FUNCTION_BLOCK FB_CO_ABERRATION
VAR_INPUT
	jd			: LREAL;		// Julian Date
	ra			: LREAL;		// RA in degrees
	dec			: LREAL; 		// Dec in degrees
	eps 		: LREAL := 0.0;
END_VAR
VAR_OUTPUT
	d_ra		: LREAL;
	d_dec		: LREAL;
END_VAR
VAR
	sunpos		: FB_SUNPOS;
	nutate		: FB_IAU2000B;
	sunra		: LREAL;
	sundec		: LREAL;
	sunlon		: LREAL;
	d_psi		: LREAL;
	d_epsilon	: LREAL; 
	eps_loc		: LREAL;		// obliquity in radians, eps or calculated if eps = 0
	t, e, peri, cd, sd, ce, te, cp, sp, cs, ss, ca, sa, term1, term2, term3, term4: LREAL;
END_VAR
VAR CONSTANT
	d2r 		: LREAL := PI/180.0;
	k			: LREAL := 20.49552; 	//constant of aberration, in arcseconds
	
END_VAR

(* https://github.com/wlandsman/IDLAstro/blob/master/pro/co_aberration.pro
;+
;  NAME:
;     CO_ABERRATION
; PURPOSE:
;     Calculate changes to Ra and Dec due to the effect of annual aberration 
; EXPLANATION:
;      as described in Meeus, Chap 23.
; CALLING SEQUENCE:
;      co_aberration, jd, ra, dec, d_ra, d_dec, [EPS = ]
; INPUTS
;       jd      : Julian Date [scalar or vector]
;       ra, dec : ra  and dec's in degrees
;
; OUTPUTS
;       d_ra, d_dec: the corrections to ra and dec due to aberration in 
;                    degrees.  (These values can be added to the true RA 
;                    and dec to get the apparent position).   Note that d_ra
;                     is *not* multiplied by cos(dec), so that 
;                     apparent_ra = ra + d_ra. 
; OPTIONAL INPUT KEYWORD:
;       eps : set this to the true obliquity of the ecliptic (in radians), or
;         it will be set for you if you don't know it (in that case, set it to
;                 an empty variable).
; NOTES:
;  These formula are from Meeus, Chapters 23.  Accuracy is much better than 1 
;   arcsecond.
;
;   The maximum deviation due to annual aberration is 20.49" and occurs when the
;   Earth velocity is perpendicular to the direction of the star.
;
; REVISION HISTORY:
;   Written, June 2002,      Chris O'Dell, U. of Wisconsin
;   Fix error with vector input   W. Landsman   June 2009
;   June 2009 update fixed case where JD was scalar but RA,Dec were vectors, but 
;     broke the case when both JD and RA,Dec were vectors Aug 2012 W. Landsman
;   Further fix when JD is 1 element vector  W. Landsman
;
;	UPDATE: HAS BEEN REWORKED FOR THE COORD STRUCTURE -> OUTPUT IS IN DEGREES
*)

T := (jd -2451545.0)/36525.0; // julian centuries from J2000 of jd.

IF eps = 0.0 THEN
	// must calculate obliquity of ecliptic
	nutate(jd := jd,
		d_psi => d_psi, 
		d_eps => d_epsilon); //d_psi and d_epsilon in arcsec
	// TRUE obliquity OF the ecliptic in radians
	eps_loc := JD2OBLIQUITY(jd, d_epsilon);
ELSE
	eps_loc := eps;
END_IF

sunpos(jd := jd, ra => sunra, dec => sundec, longmed => sunlon);

// Earth's orbital eccentricity
e := 0.016708634 - 0.000042037*T - 0.0000001267*EXPT(T, 2);
// longitude of perihelion, in degrees 
peri := 102.93735 + 1.71946*T + 0.00046*EXPT(T, 2);

//Useful Trig Functions
cd := COS(dec*d2r);		sd := SIN(dec*d2r);
ce := COS(eps_loc); 	te := TAN(eps_loc);
cp := COS(peri*d2r);	sp := SIN(peri*d2r);
cs := COS(sunlon*d2r);	ss := SIN(sunlon*d2r);
ca := COS(ra*d2r);		sa := SIN(ra*d2r);

term1 := (ca*cs*ce + sa*ss)/cd;
term2 := (ca*cp*ce + sa*sp)/cd;
term3 := (cs*ce*(te*cd - sa*sd) + ca*sd*ss);
term4 := (cp*ce*(te*cd - sa*sd) + ca*sd*sp);

d_ra := (-k * term1 + e*k * term2)/3600;
d_dec := (-k * term3 + e*k * term4)/3600;

END_FUNCTION_BLOCK

(* stored: Version 1.1.0.1, ProductVersion 3.1.4024.15
   POU FB_CO_ABERRATION: Id {78e5ea52-4364-45d1-8d65-73fef4dd6397}, SpecialFunc None *)
